Universal Robots PolyScope program: perez_FIRSTRUN.urp

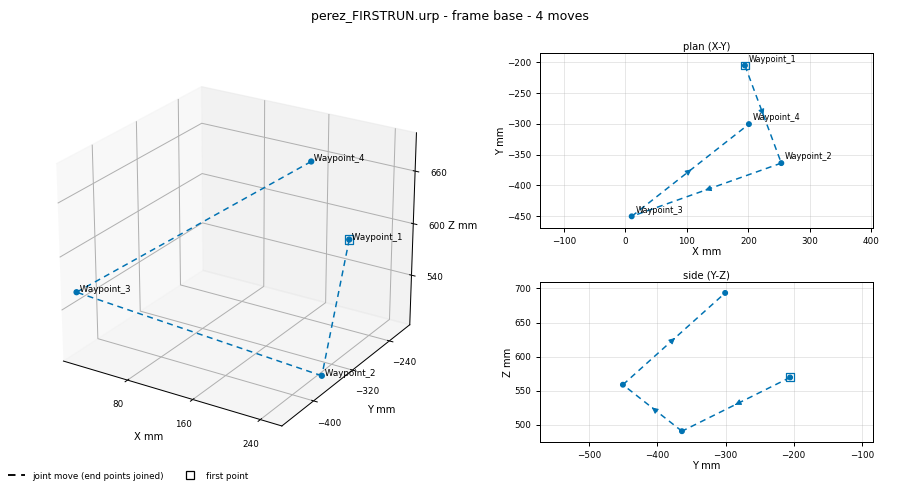
[picture p0: tool path of perez_FIRSTRUN.urp in frame base, 4 of 4 moves have a stored position in this frame; points joined in program order, loops and branches not executed]
Program perez_FIRSTRUN (createdIn=3.4.4.412 lastSavedIn=3.4.4.412 directory=/programs installation=default robotSerialNumber=2017356443)
Calibrated DH parameters: a=[0.000092, -0.116521, -0.182101, -0.000106, 0.000044, 0]; d=[0.089391, 255.189113, -82.629387, -172.449369, 0.094782, 0.082637]; alpha=[1.569598, 0.001603, 0.002015, 1.570234, -1.570307, 0]; deltaTheta=[-0.000017, 1.293309, -0.204843, -1.088417, 0.000036, -0.000078]
Robot Program (runOnlyOnce=false motionType=MoveJ speed=1.047198 acceleration=1.396263 useActiveTCP=false)
  MoveJ speed 60 deg/s, acceleration 80 deg/s^2 (useActiveTCP=false)
    Waypoint Waypoint_1: TCP in base x=194.297 y=-205.245 z=569.448 mm, rx=-2.0451 ry=2.2887 rz=-0.1925 rad; joints [-23.639, -62.275, -91.713, -107.939, 90.461, -17.296] deg
    Waypoint Waypoint_2: TCP in base x=253.457 y=-363.941 z=490.572 mm, rx=-1.2968 ry=2.8149 rz=0.0068 rad; joints [-41.102, -82.798, -88.318, -98.148, 92.33, -0.712] deg
    Waypoint Waypoint_3: TCP in base x=10.131 y=-450.529 z=558.769 mm, rx=-0.3445 ry=2.2152 rz=-1.9151 rad; joints [-74.913, -83.4, -101.709, -3.287, 92.334, -0.689] deg; flange x=10.123 y=-450.487 z=558.809 mm, rx=-0.3446 ry=2.215 rz=-1.9152 rad
    Waypoint Waypoint_4: TCP in base x=200.774 y=-300.515 z=693.44 mm, rx=-0.9024 ry=1.7845 rz=-1.5733 rad; joints [-38.943, -72.958, -90.159, -24.301, 92.328, -0.692] deg
